FUNCTION_BLOCK Saegeautomat
VAR_INPUT
END_VAR
VAR_OUTPUT
END_VAR
VAR
	//Eingänge Bedienung
	//Organisatorisches
	IN_BetriebsArt_Referenz AT %I* : BOOL;
	IN_BetriebsArt_Warmlauf AT %I* : BOOL;
	IN_BetriebsArt_Automatik AT %I* : BOOL;
	IN_BetriebsArt_Manuell AT %I* : BOOL;
	IN_Kein_Notaus AT %I* : BOOL := TRUE;
	IN_Maschine_EIN AT %I* : BOOL := TRUE;
	IN_Hydraulik_EIN AT %I* : BOOL;
	IN_Maschine_AUS AT %I* : BOOL;
	IN_Hydraulik_AUS AT %I* : BOOL;
	//Manuelle Bedienung
	IN_Kettenschmierung_Manuell_EIN AT %I* : BOOL;
	IN_Zufuehrer_Vor AT %I* : BOOL;
	IN_Zufuehrer_Rueck AT %I* : BOOL;
	IN_Stammklemmer_Oben_Hoch AT %I* : BOOL;
	IN_Stammklemmer_Oben_Runter AT %I* : BOOL;
	IN_Stammklemmer_Unten_Hoch AT %I* : BOOL;
	IN_Stammklemmer_Unten_Runter AT %I* : BOOL;
	IN_Saege_EIN AT %I* : BOOL;
	IN_Saege_AUS AT %I* : BOOL;
	IN_Saege_Hoch AT %I* : BOOL;
	IN_Saege_Runter AT %I* : BOOL;
	//Automatikmodus
	IN_Programm_Einzelsatz AT %I* : BOOL;
	IN_Zyklus_Start AT %I* : BOOL;
	IN_Zyklus_Stopp AT %I* : BOOL;
	IN_Einfache_Klemmung AT %I* : BOOL;
	
	
	//Eingänge Sensorik
	//Zuführer
	IN_Endl_Zufuehrer_Hinten AT %I* : BOOL;
	IN_Endl_Zufuehrer_Vorne AT %I* : BOOL;
	IN_Vorposition_Zufuehrer AT %I* : BOOL;
	IOL_Schaltausg_Distanzsensor_Holzende : BOOL; //Über Schaltausgang oder IO-Link Analogdaten?
	IOL_DistanzSensor_Abst : UINT;
	IN_Schaltausg_Lichtschranke AT %I* : BOOL; 
	
	//Stammklemmung Oben
	IN_Endl_Obere_Stammklemmung_Oben AT %I* : BOOL;
	IN_Endl_Obere_Stammklemmung_Unten AT %I* : BOOL;
	IN_Endl_Tastschiene AT %I* : BOOL;
	IN_Schaltausg_Druckschalter_Obere_Klemmung AT %I* : BOOL;
	//Stammklemmung Unten
	IN_Endl_Untere_Stammklemmung_Oben AT %I* : BOOL;
	IN_Endl_Untere_Stammklemmung_Unten AT %I* : BOOL;
	//Säge
	IN_Endl_Saege_Oben AT %I* : BOOL;
	IN_Endl_Saege_Unten AT %I* : BOOL;
	IN_Kettenoel_nicht_Leer AT %I* : BOOL;
	
	//Ausgänge
	//Ausgänge Hydraulik
	
	//Ausgänge Schalten
	OUT_Hydraulikpumpe_EIN AT %Q* : BOOL;
	//Ausgänge Daten
	
	
		
		
	//Interne Merker
	Maschine_EIN : BOOL;
	Hydraulik_EIN : BOOL;
	Referenz_gefahren : BOOL;
	Zyklus_beendet : BOOL;
	busy : BOOL;
	warten : BOOL;
	
	
	Referenzfahrt : Referenzfahrt;
	Warmlauf : Warmlauf;
	Manueller_Betrieb : Manueller_Betrieb;
	Automatikbetrieb : Automatik_Betrieb;
	Steuerung_Meldeleuchten : Meldeleuchte;
	OID200 : OID200DatenLesen;
	Ansteuerung_Ausgaenge : Ansteuerung_Ausgaenge;
	
	P_Flanke_Zyklus_Stopp : R_TRIG;
	P_Flanke_Zyklus_Start : R_TRIG;
	P_Flanke_Maschine_EIN : R_TRIG;
	

	
END_VAR

P_Flanke_Zyklus_Stopp(CLK := NOT IN_Zyklus_Stopp);
P_Flanke_Zyklus_Start(CLK := IN_Zyklus_Start);
P_Flanke_Maschine_EIN(CLK := IN_Maschine_EIN);


IF IN_Kein_Notaus AND IN_Maschine_EIN THEN
	Maschine_EIN := TRUE;
ELSIF NOT IN_Kein_Notaus OR IN_Maschine_AUS THEN
	Maschine_EIN := FALSE;
END_IF

IF Maschine_EIN AND IN_BetriebsArt_Referenz THEN
	Referenzfahrt(
		Kein_Notaus := IN_Kein_Notaus,
		Programm_Einzelsatz := IN_Programm_Einzelsatz,
		Zyklus_Start := P_Flanke_Zyklus_Start.Q,
		SFCInit := P_Flanke_Zyklus_Stopp.Q OR NOT IN_Kein_Notaus,
		SFCTipMode := IN_Programm_Einzelsatz,
		SFCTip := P_Flanke_Zyklus_Start.Q,
		Endl_Saege_Oben := NOT IN_Endl_Saege_Oben,
		Endl_Obere_Stammklemmung_Oben := NOT IN_Endl_Obere_Stammklemmung_Oben,
		Endl_Untere_Stammklemmung_Unten := NOT IN_Endl_Untere_Stammklemmung_Unten,
		Endl_Zufuehrer_Hinten := NOT IN_Endl_Zufuehrer_Hinten,
		busy := busy,
		Referenz_Gefahren := Referenz_gefahren,
		Zyklus_Beendet := Zyklus_beendet);	
END_IF

IF Maschine_EIN AND IN_BetriebsArt_Warmlauf THEN
	Warmlauf();
END_IF

IF Maschine_EIN AND IN_BetriebsArt_Manuell THEN
	Manueller_Betrieb(
		Kein_Notaus:= IN_Kein_Notaus, 
		Hydraulik_EIN:= IN_Hydraulik_EIN, 
		Hydraulik_AUS:= IN_Hydraulik_AUS, 
		Kettenschmierung_Manuell_EIN:= IN_Kettenschmierung_Manuell_EIN, 
		Zufuehrer_Vor:= IN_Zufuehrer_Vor, 
		Zufuehrer_Rueck:= IN_Zufuehrer_Rueck, 
		Stammklemmer_Oben_Hoch:= IN_Stammklemmer_Oben_Hoch, 
		Stammklemmer_Oben_Runter:= IN_Stammklemmer_Oben_Runter, 
		Stammklemmer_Unten_Hoch:= IN_Stammklemmer_Unten_Hoch, 
		Stammklemmer_Unten_Runter:= IN_Stammklemmer_Unten_Runter, 
		Saege_EIN:= IN_Saege_EIN, 
		Saege_AUS:= IN_Saege_AUS, 
		Saege_Hoch:= IN_Saege_Hoch, 
		Saege_Runter:= IN_Saege_Runter, 
		Endl_Zufuehrer_Hinten:= NOT IN_Endl_Zufuehrer_Hinten, 
		Endl_Zufuehrer_Vorne:= NOT IN_Endl_Zufuehrer_Vorne, 
		Vorposition_Zufuehrer:= NOT IN_Vorposition_Zufuehrer,  
		Endl_Obere_Stammklemmung_Oben:= NOT IN_Endl_Obere_Stammklemmung_Oben, 
		Endl_Obere_Stammklemmung_Unten:= NOT IN_Endl_Obere_Stammklemmung_Unten, 
		Endl_Tastschiene:= NOT IN_Endl_Tastschiene, 
		Schaltausg_Druckschalter_Obere_Klemmung:= NOT IN_Schaltausg_Druckschalter_Obere_Klemmung, 
		Endl_Untere_Stammklemmung_Oben:= NOT IN_Endl_Untere_Stammklemmung_Oben, 
		Endl_Untere_Stammklemmung_Unten:= NOT IN_Endl_Untere_Stammklemmung_Unten, 
		Endl_Saege_Oben:= NOT IN_Endl_Saege_Oben, 
		Endl_Saege_Unten:= NOT IN_Endl_Saege_Unten, 
		);
	
END_IF

IF Maschine_EIN AND IN_BetriebsArt_Automatik THEN
	Automatikbetrieb(
	Kein_Notaus:= IN_Kein_Notaus, 
	Zyklus_Start:= IN_Zyklus_Start, 
	Zyklus_Stopp:= NOT IN_Zyklus_Stopp, 
	Einfache_Klemmung := IN_Einfache_Klemmung,
	SFCInit:= not IN_Zyklus_Stopp, 
	SFCTip:= IN_Programm_Einzelsatz AND IN_Zyklus_Start, 
	SFCTipMode:= IN_Programm_Einzelsatz, 
	Endl_Zufuehrer_Hinten:= NOT IN_Endl_Zufuehrer_Hinten, 
	Endl_Zufuehrer_Vorne:= NOT IN_Endl_Zufuehrer_Vorne, 
	Vorposition_Zufuehrer:= NOT IN_Vorposition_Zufuehrer, 
	IOL_Schaltausg_Distanzsensor_Holzende:= NOT IN_Schaltausg_Lichtschranke, 
	IOL_DistanzSensor_Abst:= IOL_DistanzSensor_Abst, 
	Endl_Obere_Stammklemmung_Oben:= NOT IN_Endl_Obere_Stammklemmung_Oben, 
	Endl_Obere_Stammklemmung_Unten:= NOT IN_Endl_Obere_Stammklemmung_Unten, 
	Endl_Tastschiene:= IN_Endl_Tastschiene, 
	Schaltausg_Druckschalter_Obere_Klemmung:= not IN_Schaltausg_Druckschalter_Obere_Klemmung, 
	Endl_Untere_Stammklemmung_Oben:= NOT IN_Endl_Untere_Stammklemmung_Oben, 
	Endl_Untere_Stammklemmung_Unten:= NOT IN_Endl_Untere_Stammklemmung_Unten, 
	Endl_Saege_Oben:= NOT IN_Endl_Saege_Oben, 
	Endl_Saege_Unten:= NOT IN_Endl_Saege_Unten, 
	Warten_Auf_Weiterschalten=> , 
	Warten_auf_Material=> , 
	QStammklemmung_Oben_Hoch=> , 
	QStammklemmung_Oben_Runter=> , 
	QStammklemmung_Unten_Hoch=> , 
	QStammklemmung_Unten_Runter=> , 
	QSaege_Senken=> , 
	QSaege_Heben=> , 
	QHydraulikpumpe_EIN=> , 
	QZufuehrer_Antrieb_vor=> , 
	QZufuehrer_Antrieb_Rueck=> , 
	QSaege_Antrieb_Ein=> , 
	QKettenschmierung_EIN=> , 
	warten:= warten, 
	Hydraulik_EIN:= Hydraulik_EIN, 
	Zyklus_Beendet:= Zyklus_beendet);
END_IF

Ansteuerung_Ausgaenge(
	Saege_Hoch:= Referenzfahrt.Saege_Heben OR Manueller_Betrieb.QSaege_Heben OR Automatikbetrieb.QSaege_Heben, 
	Saege_Runter:= Manueller_Betrieb.QSaege_Senken OR Automatikbetrieb.QSaege_Senken, 
	Stammklemmung_Oben_Hoch:= Referenzfahrt.Stammklemmung_oben_Hoch OR Manueller_Betrieb.QStammklemmung_Oben_Hoch OR Automatikbetrieb.QStammklemmung_Oben_Hoch, 
	Stammklemmung_Oben_Runter:= Manueller_Betrieb.QStammklemmung_Oben_Runter OR Automatikbetrieb.QStammklemmung_Oben_Runter, 
	Stammklemmung_Unten_Hoch:= Manueller_Betrieb.QStammklemmung_Unten_Hoch OR Automatikbetrieb.QStammklemmung_Unten_Hoch,
	Stammklemmung_Unten_Runter:= Referenzfahrt.Stammklemmung_unten_Runter OR Manueller_Betrieb.QStammklemmung_Unten_Runter OR Automatikbetrieb.QStammklemmung_Unten_Runter,
	Saege_EIN := Manueller_Betrieb.QSaege_Antrieb_Ein OR Automatikbetrieb.QSaege_Antrieb_Ein,
	Zufuehrer_Vor := Manueller_Betrieb.QZufuehrer_Antrieb_vor OR Automatikbetrieb.QZufuehrer_Antrieb_vor,
	Zufuehrer_Rueck := Referenzfahrt.Zufuehrer_Zurueck OR Manueller_Betrieb.QZufuehrer_Antrieb_Rueck OR Automatikbetrieb.QZufuehrer_Antrieb_Rueck,
	endl_Zufuehrer_vorne := NOT IN_Endl_Zufuehrer_Vorne,
	endl_Zufuehrer_hinten := NOT IN_Endl_Zufuehrer_Hinten,
	endl_Zufuehrer_Vorpos := NOT IN_Vorposition_Zufuehrer,
	endl_Stammklemmung_Oben_Oben := NOT IN_Endl_Obere_Stammklemmung_Oben,
	endl_Stammklemmung_Oben_Unten := NOT IN_Endl_Obere_Stammklemmung_Unten,
	endl_Stammklemmung_Unten_Oben := NOT IN_Endl_Untere_Stammklemmung_Oben,
	endl_Stammklemmung_Unten_Unten := NOT IN_Endl_Untere_Stammklemmung_Unten,
	endl_Saege_Oben := NOT IN_Endl_Saege_Oben,
	endl_Saege_Unten:= NOT IN_Endl_Saege_Unten,
	kettenschmierung_EIN := Manueller_Betrieb.QKettenschmierung_EIN OR Automatikbetrieb.QSaege_Antrieb_Ein
);

OUT_Hydraulikpumpe_EIN := Manueller_Betrieb.QHydraulikpumpe_EIN OR Automatikbetrieb.QHydraulikpumpe_EIN OR Referenzfahrt.QHydraulik_EIN;

Steuerung_Meldeleuchten(
	Maschine_EIN := Maschine_EIN,
	Referenz_gefahren := Referenz_gefahren,
	Kettenschmierung_nicht_leer := IN_Kettenoel_nicht_Leer,
	Fehler_liegt_an := ,
	Busy := busy,
	Warten_auf_weiterschalten := Referenzfahrt.Warten_Auf_Weiterschalten OR FALSE, //Automatikbetrieb.Warten_Auf_Weiterschalten
	Zyklus_beendet := );


OID200(
 OID200SchaltSignal => IOL_Schaltausg_Distanzsensor_Holzende,
iOID200Dist_zu_Holz => IOL_DistanzSensor_Abst);

END_FUNCTION_BLOCK

(* stored: Version 1.1.0.1, ProductVersion 3.1.4024.16
   POU Saegeautomat: Id {fa192f54-9603-4bb0-b2e3-1b2d879bf32b}, SpecialFunc None *)
